TYPE E_TransferTrayCtrl :
(
	LeftToSlot,
    RightToSlot,
    SlotToLeft,
	SlotToRight
)USINT;
END_TYPE

(* stored: Version 1.1.0.1, ProductVersion 3.1.4024.11
   DUT E_TransferTrayCtrl: Id {b768cbb4-1e4f-4c99-8bb1-40236fcb4dba} *)
